INTERFACE I_EM_PalletConveyor

METHOD PUBLIC m_CloseDockingClamps : BOOL
END_METHOD

METHOD PUBLIC m_DockBox : BOOL
END_METHOD

METHOD PUBLIC m_OpenDockingClamps : BOOL
END_METHOD

METHOD PUBLIC m_UndockBox : BOOL
END_METHOD

PROPERTY PUBLIC p_bStaBoxAtDockedPosition : BOOL
GET
END_GET
END_PROPERTY

PROPERTY PUBLIC p_bStaBoxAtPreDockingPosition : BOOL
GET
END_GET
END_PROPERTY

PROPERTY p_bStaDockingClampsClosed : BOOL
GET
END_GET
END_PROPERTY

PROPERTY PUBLIC p_bStaDockingClampsOpened : BOOL
GET
END_GET
END_PROPERTY

PROPERTY PUBLIC p_bStaDockingDone : BOOL
GET
END_GET
END_PROPERTY

PROPERTY PUBLIC p_bStaDockingPositionFree : BOOL
GET
END_GET
END_PROPERTY

PROPERTY p_bStaUndockingDone : BOOL
GET
END_GET
END_PROPERTY

END_INTERFACE

(* stored: Version 1.1.0.1, ProductVersion 3.1.4024.12
   Itf I_EM_PalletConveyor: Id {accd63cb-de72-4de6-8162-fcc60f8e5bef}
   Method m_CloseDockingClamps: Id {4930bc8b-264c-400c-8ab4-e7447f386450}
   Method m_DockBox: Id {3904f15a-a308-4895-9a63-0f7535b37898}
   Method m_OpenDockingClamps: Id {c171c537-ea2e-4d50-ac08-a5c20192044f}
   Method m_UndockBox: Id {e9d9d6b7-8959-480c-b1d3-dd32ddf5bf66}
   Property p_bStaBoxAtDockedPosition: Id {333f2198-1678-4af3-96fd-a15e69f1a3f7}
   Get Get: Id {676e5387-e5b6-442e-ab99-531c6e4691c8}
   Property p_bStaBoxAtPreDockingPosition: Id {e3e172a6-95fa-4663-b6c9-e34a38a73ab2}
   Get Get: Id {10949b63-fc95-447e-9819-03046c9368b5}
   Property p_bStaDockingClampsClosed: Id {f2df1a09-9133-4e9c-a94c-89c3d55616c7}
   Get Get: Id {f9440d78-b9e6-48d3-93d5-aad047a75efc}
   Property p_bStaDockingClampsOpened: Id {f1f15574-f301-4778-a2a4-65a983766876}
   Get Get: Id {93798dba-7b77-4f9a-94c5-2f5567dc1333}
   Property p_bStaDockingDone: Id {861968af-e917-4af8-b32b-c539db149320}
   Get Get: Id {aca69bdd-0154-407c-bac0-ba19f7f91fd1}
   Property p_bStaDockingPositionFree: Id {afe652d5-de68-4c11-8d52-25e24ea972d1}
   Get Get: Id {609014dc-aef6-4646-9139-8f2a87d1ac62}
   Property p_bStaUndockingDone: Id {23811e33-9216-4ee9-b53f-a6dc94d13814}
   Get Get: Id {a90c07fc-4498-4a93-b368-62dd1630d327} *)
